// TwinCAT 3 PLC project PLC1
// ProjectVersion: 3.1.4024.0
// project tree:
//   DUTs/ E_CapStep.TcDUT, ST_Recipe.TcDUT
//   GVLs/ GVL_Line.TcGVL
//   POUs/ FB_AxisMove.TcPOU, FB_Capper.TcPOU, FB_Infeed.TcPOU, FB_Labeler.TcPOU, FB_RecipeHandler.TcPOU, FB_Scale.TcPOU, FB_Transfer.TcPOU, F_Throughput.TcPOU, MAIN.TcPOU

// ---- DUTs/E_CapStep.TcDUT
TYPE E_CapStep :
(
    Idle   := 0,
    Lower  := 10,
    Torque := 20,
    Raise  := 30,
    Done   := 40,
    Fault  := 99
) INT;
END_TYPE

// ---- DUTs/ST_Recipe.TcDUT
TYPE ST_Recipe :
STRUCT
    fTargetTorque : LREAL;      // Nm
    tTorqueTime   : TIME;       // longest a cap may take to reach torque
    nCapsPerTray  : UINT;
END_STRUCT
END_TYPE

// ---- GVLs/GVL_Line.TcGVL
{attribute 'qualified_only'}
VAR_GLOBAL
    bAutoMode      : BOOL;
    bResetRequest  : BOOL;
    stActiveRecipe : ST_Recipe;
    nCycleTimeMs   : UDINT;     // measured machine cycle, 0 until the first cycle completes
    nCapsDone      : UDINT;
END_VAR

// ---- POUs/FB_AxisMove.TcPOU
FUNCTION_BLOCK FB_AxisMove
VAR_INPUT
    bExecute  : BOOL;       // rising edge starts a move
    fPosition : LREAL;      // mm
END_VAR
VAR_OUTPUT
    bBusy  : BOOL;
    bDone  : BOOL;
    bError : BOOL;
END_VAR
VAR
    rtExecute : R_TRIG;
    fActual   : LREAL;
END_VAR

rtExecute(CLK := bExecute);
IF rtExecute.Q THEN
    bBusy := TRUE;
    bDone := FALSE;
    bError := FALSE;
END_IF
IF bBusy THEN
    fActual := fPosition;   // drive interface omitted: the move completes here
    bBusy := FALSE;
    bDone := TRUE;
END_IF
IF NOT bExecute THEN
    bDone := FALSE;
END_IF

END_FUNCTION_BLOCK

// ---- POUs/FB_Capper.TcPOU
FUNCTION_BLOCK FB_Capper
VAR_INPUT
    bStart     : BOOL;
    bCapSeated : BOOL;
    fTorque    : LREAL;     // Nm, from the spindle drive
END_VAR
VAR_OUTPUT
    bHeadDown  : BOOL;
    bSpindleOn : BOOL;
    bDone      : BOOL;
    bError     : BOOL;
    nErrorId   : UDINT;
END_VAR
VAR
    eStep       : E_CapStep;
    fbStepTimer : TON;
END_VAR

CASE eStep OF
    E_CapStep.Idle:
        bDone := FALSE;
        IF bStart THEN
            eStep := E_CapStep.Lower;
        END_IF

    E_CapStep.Lower:
        bHeadDown := TRUE;
        IF bCapSeated THEN
            eStep := E_CapStep.Torque;
        END_IF

    E_CapStep.Torque:
        bSpindleOn := TRUE;
        fbStepTimer(IN := TRUE, PT := GVL_Line.stActiveRecipe.tTorqueTime);
        IF fTorque >= GVL_Line.stActiveRecipe.fTargetTorque THEN
            bSpindleOn := FALSE;
            eStep := E_CapStep.Raise;
        ELSIF fbStepTimer.Q THEN
            bSpindleOn := FALSE;
            nErrorId := 16#0201;            // torque not reached in time
            eStep := E_CapStep.Fault;
        END_IF

    E_CapStep.Raise:
        bHeadDown := FALSE;
        GVL_Line.nCapsDone := GVL_Line.nCapsDone + 1;
        eStep := E_CapStep.Done;

    E_CapStep.Done:
        bDone := TRUE;
        IF NOT bStart THEN
            eStep := E_CapStep.Idle;
        END_IF

    E_CapStep.Fault:
        bError := TRUE;
        bSpindleOn := FALSE;
        bHeadDown := FALSE;
        IF GVL_Line.bResetRequest THEN
            bError := FALSE;
            nErrorId := 0;
            eStep := E_CapStep.Idle;
        END_IF
ELSE
    eStep := E_CapStep.Fault;
END_CASE

END_FUNCTION_BLOCK

// ---- POUs/FB_Infeed.TcPOU
FUNCTION_BLOCK FB_Infeed
VAR_INPUT
    bStart          : BOOL;
    bLinePressureOk : BOOL;
    bBottleSensor   : BOOL;
END_VAR
VAR_OUTPUT
    bBottleInPlace : BOOL;
    bPurgeValve    : BOOL;
END_VAR
VAR
    rtStart     : R_TRIG;
    nPurgeCount : UDINT;
END_VAR

rtStart(CLK := bStart);
IF rtStart.Q THEN
    Act_Purge();        // blow the line clear before the first bottle
END_IF
bBottleInPlace := bStart AND bBottleSensor;

ACTION Act_Purge:
REPEAT
    bPurgeValve := TRUE;
    nPurgeCount := nPurgeCount + 1;
UNTIL bLinePressureOk
END_REPEAT
bPurgeValve := FALSE;
END_ACTION

END_FUNCTION_BLOCK

// ---- POUs/FB_Labeler.TcPOU
FUNCTION_BLOCK FB_Labeler
VAR_INPUT
    nLabels : UDINT;
    pRoll   : POINTER TO UDINT;     // remaining labels on the roll, from the HMI
END_VAR
VAR_OUTPUT
    nRollsUsed : UDINT;
    bRollLow   : BOOL;
END_VAR
VAR CONSTANT
    cLabelsPerRoll : UDINT := 2000;
END_VAR

nRollsUsed := nLabels / cLabelsPerRoll;
IF pRoll <> 0 THEN
    bRollLow := pRoll^ < 100;
END_IF

END_FUNCTION_BLOCK

// ---- POUs/FB_RecipeHandler.TcPOU
FUNCTION_BLOCK FB_RecipeHandler
VAR_INPUT
    pSource : POINTER TO ST_Recipe;     // set by the HMI when a recipe is selected
END_VAR

METHOD Apply : BOOL
GVL_Line.stActiveRecipe := pSource^;
Apply := TRUE;
END_METHOD

END_FUNCTION_BLOCK

// ---- POUs/FB_Scale.TcPOU
FUNCTION_BLOCK FB_Scale
VAR_INPUT
    nRaw : DINT;            // counts from the load cell terminal
END_VAR
VAR
    fWeight     : LREAL;    // g
    fLastWeight : LREAL;
END_VAR

fLastWeight := fWeight;
fWeight := DINT_TO_LREAL(nRaw) * 0.01;

PROPERTY IsSettled : BOOL
GET
IsSettled := (fWeight = fLastWeight);
END_GET
END_PROPERTY

END_FUNCTION_BLOCK

// ---- POUs/FB_Transfer.TcPOU
FUNCTION_BLOCK FB_Transfer
VAR_INPUT
    bRequest : BOOL;
    fTarget  : LREAL;       // mm
END_VAR
VAR_OUTPUT
    bInPosition : BOOL;
END_VAR
VAR
    fbMove : FB_AxisMove;
END_VAR

IF bRequest THEN
    fbMove(bExecute := TRUE, fPosition := fTarget);
END_IF
bInPosition := fbMove.bDone;

END_FUNCTION_BLOCK

// ---- POUs/F_Throughput.TcPOU
FUNCTION F_Throughput : UDINT
VAR_INPUT
    nCaps        : UDINT;
    nCycleTimeMs : UDINT;
END_VAR

F_Throughput := nCaps * 60000 / nCycleTimeMs;

END_FUNCTION

// ---- POUs/MAIN.TcPOU
PROGRAM MAIN
VAR
    fbInfeed   : FB_Infeed;
    fbCapper   : FB_Capper;
    fbTransfer : FB_Transfer;
    fbScale    : FB_Scale;
    fbRecipe   : FB_RecipeHandler;
    fbLabeler  : FB_Labeler;
    nPerMinute : UDINT;
END_VAR

fbInfeed(bStart := GVL_Line.bAutoMode);
fbCapper(bStart := fbInfeed.bBottleInPlace);
fbTransfer(bRequest := fbCapper.bDone, fTarget := 250.0);
fbScale();
fbLabeler(nLabels := GVL_Line.nCapsDone);
nPerMinute := F_Throughput(nCaps := GVL_Line.nCapsDone,
                           nCycleTimeMs := GVL_Line.nCycleTimeMs);

END_PROGRAM
